TYPE FLOWMETER_VALUES :
STRUCT
	MassFlow:REAL;
	VolumeFlow:REAL;
	CorrectedVolueFLow:REAL;
	Density:REAL;
	ReferenceDensity:REAL;
	Temperature:REAL;
	TotalMass:REAL;
END_STRUCT
END_TYPE

(* stored: Version 1.1.0.1, ProductVersion 3.1.0.26
   DUT FLOWMETER_VALUES: Id {48aaf078-15a9-418d-8042-99b2d4f6d6b4} *)
